Yaskawa INFORM job: R2_72,2(0,0).JBI

/JOB
//NAME R2_72,2(0,0)
///FOLDERNAME KR_OK
//POS
///NPOS 41,41,0,2,0,0
///TOOL 0
///POSTYPE PULSE
///PULSE
C00000=120729,38464,-23607,67702,92694,37114
C00001=120728,81583,44137,67576,84483,28591
C00002=120728,81594,44149,67576,84482,28590
C00003=120728,81598,44155,67576,84481,28590
C00004=121074,78743,40667,67457,84531,28927
C00005=121609,78761,40687,67335,84187,28996
C00006=120728,81586,44140,67576,84482,28591
C00007=120728,81598,44155,67576,84481,28590
C00008=120728,81620,44182,67577,84479,28587
C00009=120728,81940,45939,67638,84105,28196
C00010=120728,81620,44182,67577,84479,28587
C00011=120728,81598,44155,67576,84481,28590
C00012=120728,82318,42212,50838,72434,30029
C00013=120728,81757,44308,51214,71418,29445
C00014=120728,83572,46546,51324,71133,29280
C00015=120728,81757,44308,51214,71418,29445
C00016=120728,82318,42212,50838,72434,30029
C00017=120728,82410,41725,50759,72659,30157
C00018=120728,82684,40958,50622,73056,30381
C00019=120728,83470,39162,50303,74040,30931
C00020=120731,108704,30437,520,103146,-53106
C00021=120730,95364,30685,507,96140,-53135
C00022=120729,92856,31465,505,94371,-53142
C00023=120902,90721,30804,453,93677,-53092
C00024=120076,91948,31897,698,93643,-53342
C00025=120729,92386,31163,506,94315,-53143
C00026=120890,97827,39416,458,92029,-53101
C00027=121108,130065,79645,455,95365,-53013
C00028=120821,132587,79324,499,96860,-53101
C00029=120730,97149,30254,16854,109142,-86058
C00030=94374,59905,-24624,-6692,95808,-73268
C00031=94859,43835,-17383,-4554,74801,-71238
C00032=94859,41415,-16000,-4599,72712,-71159
C00033=88904,46834,-10813,7148,76662,-70087
C00034=94590,38531,-17304,-4457,72022,-71215
C00035=94826,41033,-16151,-4582,72608,-71165
C00036=90359,45192,-12541,6368,76777,-69648
C00037=101841,55528,-4022,-16346,83094,-70723
C00038=102455,61397,2318,-16651,82349,-70435
C00039=102039,71942,670,-16368,88461,-71374
C00040=48492,61943,-11432,-541,72797,-1948
BC00000=247969,284149,1069855
BC00001=247969,284149,1069855
BC00002=242395,281084,1053929
BC00003=240166,279858,1047559
BC00004=240163,279216,1029407
BC00005=240163,279216,1029407
BC00006=240163,279216,1029407
BC00007=240166,279858,1047559
BC00008=234047,281783,1046735
BC00009=234047,281783,1046735
BC00010=234047,281783,1046735
BC00011=240166,279858,1047559
BC00012=204016,317970,1075175
BC00013=204014,317334,1075175
BC00014=204014,317334,1075175
BC00015=204014,317334,1075175
BC00016=204016,317970,1075175
BC00017=217547,308995,1075175
BC00018=218903,310893,1075175
BC00019=222293,315638,1075175
BC00020=148834,300449,1075175
BC00021=148876,300454,1075175
BC00022=146152,298931,1075175
BC00023=145063,298322,1075175
BC00024=145063,298322,1075175
BC00025=145063,298322,1075175
BC00026=145063,298322,1075175
BC00027=145063,298322,1075175
BC00028=145063,298322,1075175
BC00029=163962,261690,1075175
BC00030=16042,269075,1075175
BC00031=16207,275422,1075175
BC00032=16871,271934,1075175
BC00033=17137,270539,1075175
BC00034=17137,270539,1075175
BC00035=17137,270539,1075175
BC00036=17137,270539,1075175
BC00037=17137,270539,1075175
BC00038=17137,270539,1075175
BC00039=17137,270539,1075175
BC00040=49225,325633,1075175
///POSTYPE BASE
///RECTAN
///RCONF 0,0,0,0,0,0,0,0,0,0,0,0,0,0,0,0,0,0,0,0,0,0,0,0
P00006=0.222,-3.123,-1.508,0.0000,0.0000,0.0000
P00021=-0.225,-6.128,-0.405,0.0000,0.0000,0.0000
//INST
///DATE 2023/11/16 10:51
///ATTR SC,RW
///GROUP1 RB1,BS1
NOP
'R2_72.2(0,0)
'Path S1184
SFTOF
MOVJ C00000 BC00000 VJ=20.00
MOVJ C00001 BC00001 VJ=20.00
MOVL C00002 BC00002 V=100.0
MOVL C00003 BC00003 V=100.0
MOVL C00004 BC00004 V=60.0
REFP 3 C00005 BC00005
CALL JOB:SEARCH-R1
SET P021 P006
SFTON P021
MOVL C00006 BC00006 V=60.0
MOVL C00007 BC00007 V=100.0
MOVL C00008 BC00008 V=60.0
REFP 3 C00009 BC00009
CALL JOB:SEARCH-R1
SET P021 P006
SFTON P021
MOVL C00010 BC00010 V=60.0
MOVL C00011 BC00011 V=100.0
MOVL C00012 BC00012 V=100.0
MOVL C00013 BC00013 V=60.0
REFP 3 C00014 BC00014
CALL JOB:SEARCH-R1
SET P021 P006
SFTON P021
MOVL C00015 BC00015 V=60.0
MOVL C00016 BC00016 V=100.0
MOVL C00017 BC00017 V=100.0
MOVL C00018 BC00018 V=100.0
MOVL C00019 BC00019 V=100.0
'Path W1186
SFTOF
SFTON P021
MOVJ C00020 BC00020 VJ=20.00
MOVJ C00021 BC00021 VJ=20.00
MOVL C00022 BC00022 V=100.0
MOVL C00023 BC00023 V=100.0 PL=0
REFP 1 C00024 BC00024
REFP 2 C00025 BC00025
MACRO1 MJ#(0) ARGF6
ARCON
MOVL C00026 BC00026 V=11.7
MOVL C00027 BC00027 V=11.7
ARCOF
MOVL C00028 BC00028 V=100.0
MOVL C00029 BC00029 V=100.0
SFTOF
'Path W1188
SFTOF
SFTON P021
MOVJ C00030 BC00030 VJ=20.00
MOVJ C00031 BC00031 VJ=20.00
MOVJ C00032 BC00032 VJ=20.00
MOVL C00033 BC00033 V=100.0 PL=0
REFP 1 C00034 BC00034
REFP 2 C00035 BC00035
MACRO1 MJ#(0) ARGF6
ARCON
MOVL C00036 BC00036 V=11.7
MOVL C00037 BC00037 V=11.7
MOVL C00038 BC00038 V=11.7
ARCOF
MOVL C00039 BC00039 V=100.0
MOVJ C00040 BC00040 VJ=20.00
SFTOF
END
